TYPE EL2809_PDOS :
	STRUCT
		
		PlcToHw : EL2809_PLCTOHW_PDOS;
		
	END_STRUCT
END_TYPE

(* stored: Version 1.1.0.1
   DUT EL2809_PDOS: Id {87eab8a9-1930-4725-bc76-34cc289bb9c0} *)
